{attribute 'enable_dynamic_creation'}
FUNCTION_BLOCK FB_Wait EXTENDS FB_BaseAction
VAR
	// Wait specific properties
	duration : TIME;
	elapsedTime : TIME;
END_VAR

// Wait implementation

END_FUNCTION_BLOCK

(* stored: Version 1.1.0.1
   POU FB_Wait: Id {f1b2c3d4-7774-7777-7777-777777777777} *)
